FUNCTION_BLOCK GripperPneumatic (* Basic Function Block Type *)
  (* Standard: 61499-2 *)
  (* Version 0.0, 2014-08-21, 4DIAC-IDE, 4DIAC-Consortium *)
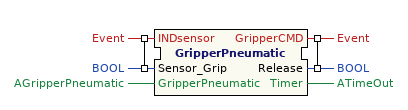
  EVENT_INPUT
    INDsensor WITH Sensor_Grip;
  END_EVENT
  EVENT_OUTPUT
    GripperCMD WITH Release;
  END_EVENT
  VAR_INPUT
    Sensor_Grip : BOOL; (* Input event qualifier *)
  END_VAR
  VAR_OUTPUT
    Release : BOOL; (* Output event qualifier *)
  END_VAR
  SOCKETS
    GripperPneumatic : AGripperPneumatic;
  END_SOCKETS
  PLUGS
    Timer : ATimeOut;
  END_PLUGS
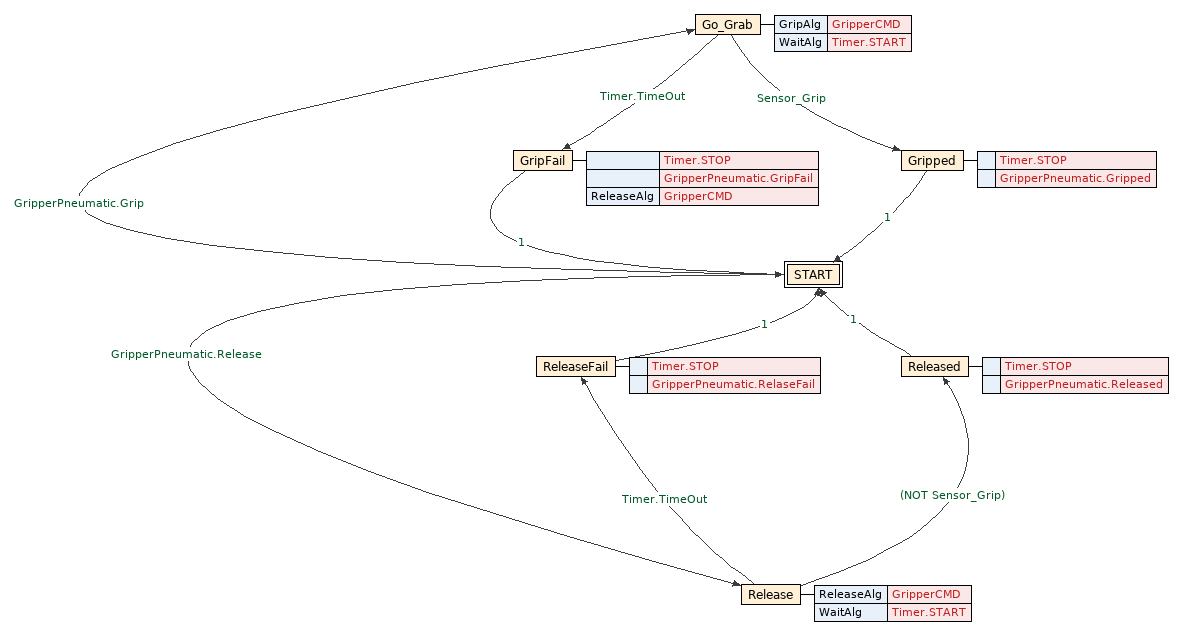
  EC_STATES
    START; (* Initial State *)
    Released : -> Timer.STOP, -> GripperPneumatic.Released;
    Release : ReleaseAlg -> GripperCMD, WaitAlg -> Timer.START;
    Gripped : -> Timer.STOP, -> GripperPneumatic.Gripped;
    Go_Grab : GripAlg -> GripperCMD, WaitAlg -> Timer.START;
    GripFail : -> Timer.STOP, -> GripperPneumatic.GripFail, ReleaseAlg -> GripperCMD;
    ReleaseFail : -> Timer.STOP, -> GripperPneumatic.RelaseFail;
  END_STATES
  EC_TRANSITIONS
    START TO Go_Grab := GripperPneumatic.Grip;
    START TO Release := GripperPneumatic.Release;
    Release TO ReleaseFail := Timer.TimeOut;
    Go_Grab TO GripFail := Timer.TimeOut;
    Go_Grab TO Gripped := Sensor_Grip;
    Release TO Released := (NOT Sensor_Grip);
    Gripped TO START := 1;
    ReleaseFail TO START := 1;
    GripFail TO START := 1;
    Released TO START := 1;
  END_TRANSITIONS
  ALGORITHM GripAlg IN ST:
Release := TRUE;
  END_ALGORITHM
  ALGORITHM ReleaseAlg IN ST:
Release:= FALSE;
  END_ALGORITHM
  ALGORITHM WaitAlg IN ST: (* Timedelay for sensor data *)
Timer.DT:= T#5s;
  END_ALGORITHM
  (* Service FB interface/Run time: Basic Function Block Type *)
END_FUNCTION_BLOCK
